{attribute 'Tc2GvlVarNames'}
(* Generated automatically by TwinCAT - (read only) *)
VAR_CONFIG
	.Main_Relais AT %QX6.0 : BOOL;	(*  ~ {LinkedWith:TIID^Gerät 4 (RT-Ethernet)^Box 1 (BK9000 192.168.100.5)^Klemme 24 (KL2012)^Kanal 2^Ausgang} *)
	.Feedback_Mainswitch AT %IX154.0 : BOOL;	(*  ~ {LinkedWith:TIID^Gerät 4 (RT-Ethernet)^Box 1 (BK9000 192.168.100.5)^Klemme 19 (KL1104)^Kanal 1^Eingang} *)
	.OUT_Mainswitch AT %QX6.1 : BOOL;	(*  ~ {LinkedWith:TIID^Gerät 4 (RT-Ethernet)^Box 1 (BK9000 192.168.100.5)^Klemme 24 (KL2012)^Kanal 1^Ausgang} *)
	.VDC_24_OK AT %IX154.1 : BOOL;	(*  ~ {LinkedWith:TIID^Gerät 4 (RT-Ethernet)^Box 1 (BK9000 192.168.100.5)^Klemme 19 (KL1104)^Kanal 2^Eingang} *)
	.Sollwert_OUT_NV AT %QB20 : INT;
	.Istwert_IN_NV AT %IB176 : INT;
	.Temp_Heatmatt1_IN AT %IB48 : INT;	(*  ~ {LinkedWith:TIID^Gerät 5 (EtherCAT)^Sensorbox_eingänge^Klemme 24 (EL3314)^TC Inputs Channel 1^Value} *)
	.Temp_Heatmatt2_IN AT %IB50 : INT;	(*  ~ {LinkedWith:TIID^Gerät 5 (EtherCAT)^Sensorbox_eingänge^Klemme 24 (EL3314)^TC Inputs Channel 3^Value} *)
	.Temp_Heatmatt3_IN AT %IB52 : INT;	(*  ~ {LinkedWith:TIID^Gerät 5 (EtherCAT)^Sensorbox_eingänge^Klemme 25 (EL3314)^TC Inputs Channel 2^Value} *)
	.Temp_Heatmatt4_IN AT %IB54 : INT;	(*  ~ {LinkedWith:TIID^Gerät 5 (EtherCAT)^Sensorbox_eingänge^Klemme 25 (EL3314)^TC Inputs Channel 4^Value} *)
	.Temp_Heatmatt5_IN AT %IB56 : INT;	(*  ~ {LinkedWith:TIID^Gerät 5 (EtherCAT)^Sensorbox_eingänge^Klemme 25 (EL3314)^TC Inputs Channel 3^Value} *)
	.Temp_Heatmatt6_IN AT %IB58 : INT;	(*  ~ {LinkedWith:TIID^Gerät 5 (EtherCAT)^Sensorbox_eingänge^Klemme 25 (EL3314)^TC Inputs Channel 1^Value} *)
	.Temp_Heatmatt7_IN AT %IB60 : INT;	(*  ~ {LinkedWith:TIID^Gerät 5 (EtherCAT)^Sensorbox_eingänge^Klemme 24 (EL3314)^TC Inputs Channel 2^Value} *)
	.Temp_Heatmatt8_IN AT %IB62 : INT;	(*  ~ {LinkedWith:TIID^Gerät 5 (EtherCAT)^Sensorbox_eingänge^Klemme 24 (EL3314)^TC Inputs Channel 4^Value} *)
	.Temp_Heatmatt9_IN AT %IB64 : INT;	(*  ~ {LinkedWith:TIID^Gerät 5 (EtherCAT)^Sensorbox_eingänge^Klemme 26 (EL3314)^TC Inputs Channel 1^Value} *)
	.Temp_Heatmatt10_IN AT %IB66 : INT;	(*  ~ {LinkedWith:TIID^Gerät 5 (EtherCAT)^Sensorbox_eingänge^Klemme 26 (EL3314)^TC Inputs Channel 2^Value} *)
	.Current_IN_HEAT_Reg_1 AT %IB74 : INT;	(*  ~ {LinkedWith:TIID^Gerät 4 (RT-Ethernet)^Box 1 (BK9000 192.168.100.5)^Klemme 31 (KL3054)^Kanal 2^Daten Ein} *)
	.Current_IN_HEAT_Reg_2 AT %IB76 : INT;	(*  ~ {LinkedWith:TIID^Gerät 4 (RT-Ethernet)^Box 1 (BK9000 192.168.100.5)^Klemme 31 (KL3054)^Kanal 3^Daten Ein} *)
	.Current_IN_HEAT_Reg_3 AT %IB78 : INT;	(*  ~ {LinkedWith:TIID^Gerät 4 (RT-Ethernet)^Box 1 (BK9000 192.168.100.5)^Klemme 31 (KL3054)^Kanal 4^Daten Ein} *)
	.Current_IN_HEAT_Reg_4 AT %IB80 : INT;
	.Current_IN_Compressor_L1 AT %IB82 : INT;	(*  ~ {LinkedWith:TIID^Gerät 4 (RT-Ethernet)^Box 1 (BK9000 192.168.100.5)^Klemme 28 (KL3022)^Kanal 1^Daten Ein} *)
	.Current_IN_Compressor_L2 AT %IB84 : INT;	(*  ~ {LinkedWith:TIID^Gerät 4 (RT-Ethernet)^Box 1 (BK9000 192.168.100.5)^Klemme 28 (KL3022)^Kanal 2^Daten Ein} *)
	.Current_IN_Compressor_L3 AT %IB86 : INT;	(*  ~ {LinkedWith:TIID^Gerät 4 (RT-Ethernet)^Box 1 (BK9000 192.168.100.5)^Klemme 29 (KL3022)^Kanal 1^Daten Ein} *)
	.Current_IN_SteamFan_L1 AT %IB88 : INT;	(*  ~ {LinkedWith:TIID^Gerät 4 (RT-Ethernet)^Box 1 (BK9000 192.168.100.5)^Klemme 30 (KL3054)^Kanal 3^Daten Ein} *)
	.Current_IN_SteamFan_L2 AT %IB90 : INT;	(*  ~ {LinkedWith:TIID^Gerät 4 (RT-Ethernet)^Box 1 (BK9000 192.168.100.5)^Klemme 30 (KL3054)^Kanal 4^Daten Ein} *)
	.Current_IN_SteamFan_L3 AT %IB92 : INT;	(*  ~ {LinkedWith:TIID^Gerät 4 (RT-Ethernet)^Box 1 (BK9000 192.168.100.5)^Klemme 31 (KL3054)^Kanal 1^Daten Ein} *)
	.Current_IN_Fan_L1 AT %IB94 : INT;
	.Current_IN_Fan_L2 AT %IB96 : INT;
	.Current_IN_Fan_L3 AT %IB98 : INT;
	.Current_IN_Complete_L1 AT %IB100 : INT;	(*  ~ {LinkedWith:TIID^Gerät 4 (RT-Ethernet)^Box 1 (BK9000 192.168.100.5)^Klemme 26 (KL3022)^Kanal 2^Daten Ein} *)
	.Current_IN_Complete_L2 AT %IB102 : INT;	(*  ~ {LinkedWith:TIID^Gerät 4 (RT-Ethernet)^Box 1 (BK9000 192.168.100.5)^Klemme 27 (KL3022)^Kanal 1^Daten Ein} *)
	.Current_IN_Complete_L3 AT %IB104 : INT;	(*  ~ {LinkedWith:TIID^Gerät 4 (RT-Ethernet)^Box 1 (BK9000 192.168.100.5)^Klemme 27 (KL3022)^Kanal 2^Daten Ein} *)
	.Compressor_ON AT %QX6.2 : BOOL;	(*  ~ {LinkedWith:TIID^Gerät 4 (RT-Ethernet)^Box 1 (BK9000 192.168.100.5)^Klemme 23 (KL2012)^Kanal 1^Ausgang} *)
	.Compressor_Switch_ON AT %QX6.3 : BOOL;	(*  ~ {LinkedWith:TIID^Gerät 4 (RT-Ethernet)^Box 1 (BK9000 192.168.100.5)^Klemme 21 (KL2114)^Kanal 1^Ausgang} *)
	.Compressor_OK AT %IX154.2 : BOOL;	(*  ~ {LinkedWith:TIID^Gerät 4 (RT-Ethernet)^Box 1 (BK9000 192.168.100.5)^Klemme 20 (KL1104)^Kanal 2^Eingang} *)
	.Compressor_Circuit_breaker AT %IX154.3 : BOOL;	(*  ~ {LinkedWith:TIID^Gerät 4 (RT-Ethernet)^Box 1 (BK9000 192.168.100.5)^Klemme 20 (KL1104)^Kanal 1^Eingang} *)
	.Compressor_Setpoint_OUT AT %QB0 : INT;	(*  ~ {LinkedWith:TIID^Gerät 4 (RT-Ethernet)^Box 1 (BK9000 192.168.100.5)^Klemme 32 (KL4002)^Kanal 1^Daten Aus} *)
	.Compressor_Actual_Turn_IN AT %IB144 : INT;	(*  ~ {LinkedWith:TIID^Gerät 4 (RT-Ethernet)^Box 1 (BK9000 192.168.100.5)^Klemme 25 (KL3022)^Kanal 1^Daten Ein} *)
	.Compressor_PT100_value AT %IB146 : INT;	(*  ~ {LinkedWith:TIID^Gerät 5 (EtherCAT)^Heizbox^Klemme 10 (EL3214)^RTD Inputs Channel 1^Value} *)
	.Compressor_PT100_error AT %IX154.4 : BOOL;	(*  ~ {LinkedWith:TIID^Gerät 5 (EtherCAT)^Heizbox^Klemme 10 (EL3214)^RTD Inputs Channel 1^Status^Error} *)
	.Fan_ON AT %QX32.0 : BOOL;	(*  ~ {LinkedWith:TIID^Gerät 4 (RT-Ethernet)^Box 1 (BK9000 192.168.100.5)^Klemme 21 (KL2114)^Kanal 4^Ausgang} *)
	.Fan_OK AT %IX154.5 : BOOL;	(*  ~ {LinkedWith:TIID^Gerät 4 (RT-Ethernet)^Box 1 (BK9000 192.168.100.5)^Klemme 20 (KL1104)^Kanal 3^Eingang} *)
	.Setpoint_Fan_OUT AT %QB2 : INT;	(*  ~ {LinkedWith:TIID^Gerät 4 (RT-Ethernet)^Box 1 (BK9000 192.168.100.5)^Klemme 32 (KL4002)^Kanal 2^Daten Aus} *)
	.Fan_Actual_Turn_IN AT %IB148 : INT;	(*  ~ {LinkedWith:TIID^Gerät 4 (RT-Ethernet)^Box 1 (BK9000 192.168.100.5)^Klemme 25 (KL3022)^Kanal 2^Daten Ein} *)
	.FAN_Switch_ON AT %QX6.5 : BOOL;	(*  ~ {LinkedWith:TIID^Gerät 4 (RT-Ethernet)^Box 1 (BK9000 192.168.100.5)^Klemme 21 (KL2114)^Kanal 2^Ausgang} *)
	.SteamFan_ON AT %QX6.6 : BOOL;	(*  ~ {LinkedWith:TIID^Gerät 4 (RT-Ethernet)^Box 1 (BK9000 192.168.100.5)^Klemme 22 (KL2114)^Kanal 3^Ausgang} *)
	.Setpoint_SteamFan_OUT AT %QB4 : INT;	(*  ~ {LinkedWith:TIID^Gerät 4 (RT-Ethernet)^Box 1 (BK9000 192.168.100.5)^Klemme 33 (KL4002)^Kanal 1^Daten Aus} *)
	.SteamFan_Actual_Turn_IN AT %IB150 : INT;	(*  ~ {LinkedWith:TIID^Gerät 4 (RT-Ethernet)^Box 1 (BK9000 192.168.100.5)^Klemme 26 (KL3022)^Kanal 1^Daten Ein} *)
	.SteamFAN_Switch_ON AT %QX6.7 : BOOL;	(*  ~ {LinkedWith:TIID^Gerät 4 (RT-Ethernet)^Box 1 (BK9000 192.168.100.5)^Klemme 21 (KL2114)^Kanal 3^Ausgang} *)
	.SteamFan_PTC_IN AT %IX154.7 : BOOL;	(*  ~ {LinkedWith:TIID^Gerät 5 (EtherCAT)^Klemme 41 (EK1200)^Klemme 3 (EL1382)^Channel 1^Input} *)
	.SteamFan_PTC_Error AT %IX155.0 : BOOL;	(*  ~ {LinkedWith:TIID^Gerät 5 (EtherCAT)^Klemme 41 (EK1200)^Klemme 3 (EL1382)^Channel 1^Error} *)
	.Heizelement_Auffangbecken_Mainswitch AT %QX8.4 : BOOL;	(*  ~ {LinkedWith:TIID^Gerät 4 (RT-Ethernet)^Box 1 (BK9000 192.168.100.5)^Klemme 22 (KL2114)^Kanal 1^Ausgang} *)
	.Heat_matt1 AT %QX9.0 : BOOL;	(*  ~ {LinkedWith:TIID^Gerät 5 (EtherCAT)^Sensorbox_Relais^Box 54 (BK1250)^Klemme 7 (KL2631)^Kanal 1^Ausgang} *)
	.Heat_matt2 AT %QX9.1 : BOOL;	(*  ~ {LinkedWith:TIID^Gerät 5 (EtherCAT)^Sensorbox_Relais^Box 54 (BK1250)^Klemme 8 (KL2631)^Kanal 1^Ausgang} *)
	.Heat_matt3 AT %QX9.2 : BOOL;	(*  ~ {LinkedWith:TIID^Gerät 5 (EtherCAT)^Sensorbox_Relais^Box 54 (BK1250)^Klemme 9 (KL2631)^Kanal 1^Ausgang} *)
	.Heat_matt4 AT %QX9.3 : BOOL;	(*  ~ {LinkedWith:TIID^Gerät 5 (EtherCAT)^Sensorbox_Relais^Box 54 (BK1250)^Klemme 10 (KL2631)^Kanal 1^Ausgang} *)
	.Heat_matt5 AT %QX9.4 : BOOL;	(*  ~ {LinkedWith:TIID^Gerät 5 (EtherCAT)^Sensorbox_Relais^Box 54 (BK1250)^Klemme 12 (KL2631)^Kanal 1^Ausgang} *)
	.Heat_matt6 AT %QX9.5 : BOOL;	(*  ~ {LinkedWith:TIID^Gerät 5 (EtherCAT)^Sensorbox_Relais^Box 54 (BK1250)^Klemme 13 (KL2631)^Kanal 1^Ausgang} *)
	.Heat_matt7 AT %QX9.6 : BOOL;	(*  ~ {LinkedWith:TIID^Gerät 5 (EtherCAT)^Sensorbox_Relais^Box 54 (BK1250)^Klemme 14 (KL2631)^Kanal 1^Ausgang} *)
	.Heat_matt8 AT %QX9.7 : BOOL;	(*  ~ {LinkedWith:TIID^Gerät 5 (EtherCAT)^Sensorbox_Relais^Box 54 (BK1250)^Klemme 15 (KL2631)^Kanal 1^Ausgang} *)
	.Heat_matt9 AT %QX10.0 : BOOL;	(*  ~ {LinkedWith:TIID^Gerät 5 (EtherCAT)^Sensorbox_eingänge^Klemme 18 (EL2828)^Channel 6^Output} *)
	.Heat_matt10 AT %QX10.1 : BOOL;	(*  ~ {LinkedWith:TIID^Gerät 5 (EtherCAT)^Sensorbox_eingänge^Klemme 18 (EL2828)^Channel 7^Output} *)
	.HEAT_Reg_Mainswitch_OUT AT %QX10.6 : BOOL;	(*  ~ {LinkedWith:TIID^Gerät 4 (RT-Ethernet)^Box 1 (BK9000 192.168.100.5)^Klemme 22 (KL2114)^Kanal 2^Ausgang} *)
	.HEAT_Reg_1_OUT AT %QX10.2 : BOOL;	(*  ~ {LinkedWith:TIID^Gerät 5 (EtherCAT)^Heizbox^Klemme 7 (EL2828)^Channel 1^Output} *)
	.HEAT_Reg_2_OUT AT %QX10.3 : BOOL;	(*  ~ {LinkedWith:TIID^Gerät 5 (EtherCAT)^Heizbox^Klemme 7 (EL2828)^Channel 2^Output} *)
	.HEAT_Reg_3_OUT AT %QX10.4 : BOOL;	(*  ~ {LinkedWith:TIID^Gerät 5 (EtherCAT)^Heizbox^Klemme 7 (EL2828)^Channel 7^Output} *)
	.HEAT_Reg_4_OUT AT %QX10.5 : BOOL;	(*  ~ {LinkedWith:TIID^Gerät 5 (EtherCAT)^Heizbox^Klemme 7 (EL2828)^Channel 8^Output} *)
	.Heat_matt_Group1_1_4_manu AT %QX12.0 : BOOL;	(*  ~ {LinkedWith:TIID^Gerät 5 (EtherCAT)^Sensorbox_eingänge^Klemme 18 (EL2828)^Channel 1^Output} *)
	.Heat_matt_Group2_5_8_manu AT %QX12.1 : BOOL;	(*  ~ {LinkedWith:TIID^Gerät 5 (EtherCAT)^Sensorbox_eingänge^Klemme 18 (EL2828)^Channel 2^Output} *)
	.Heat_matt_Group3_9_10_manu AT %QX12.2 : BOOL;	(*  ~ {LinkedWith:TIID^Gerät 5 (EtherCAT)^Sensorbox_eingänge^Klemme 18 (EL2828)^Channel 3^Output} *)
	.LED_RED_OUT AT %QX11.1 : BOOL;	(*  ~ {LinkedWith:TIID^Gerät 5 (EtherCAT)^Sensorbox_eingänge^Klemme 19 (EL2828)^Channel 3^Output} *)
	.LED_green_OUT AT %QX11.2 : BOOL;	(*  ~ {LinkedWith:TIID^Gerät 5 (EtherCAT)^Sensorbox_eingänge^Klemme 19 (EL2828)^Channel 1^Output} *)
	.LED_yellow_OUT AT %QX11.3 : BOOL;	(*  ~ {LinkedWith:TIID^Gerät 5 (EtherCAT)^Sensorbox_eingänge^Klemme 19 (EL2828)^Channel 2^Output} *)
	.LED_white_OUT AT %QX11.4 : BOOL;	(*  ~ {LinkedWith:TIID^Gerät 5 (EtherCAT)^Sensorbox_eingänge^Klemme 19 (EL2828)^Channel 4^Output} *)
END_VAR

(* stored: Version 1.1.0.1, ProductVersion 3.1.4020.6
   GVL TwinCAT_Configuration: Id {dda5512a-45d5-4a62-8cf2-55c7e8d8afb6} *)
